// TIA Portal V18 export
VAR_GLOBAL   // PLC tag table "Default tag table"
   MOTOR_OUTPUT AT %M0.0 : Bool;
   MOTOR_START AT %M0.1 : Bool;
   MOTOR_STOP AT %M0.2 : Bool;
END_VAR
